FUNCTION_BLOCK integEC (* Basic Function Block Type *)
  (* Standard: 61499-2 *)
  (* Version 0.0, 2007-06-14, milos, nxtControl GmbH, Template *)
  PACKAGE Main;
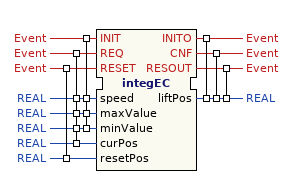
  EVENT_INPUT
    INIT WITH speed, maxValue, minValue; (* Initialization Request *)
    REQ WITH speed, maxValue, minValue, curPos; (* cycle calculation call *)
    RESET WITH resetPos;
  END_EVENT
  EVENT_OUTPUT
    INITO WITH liftPos; (* Initialization Confirm *)
    CNF WITH liftPos; (* Execution Confirmation *)
    RESOUT WITH liftPos;
  END_EVENT
  VAR_INPUT
    speed : REAL := 0.0; (* pv1 to integrate *)
    maxValue : REAL;
    minValue : REAL;
    curPos : REAL;
    resetPos : REAL;
  END_VAR
  VAR_OUTPUT
    liftPos : REAL := 0.0; (* out value (depends on integType) *)
  END_VAR
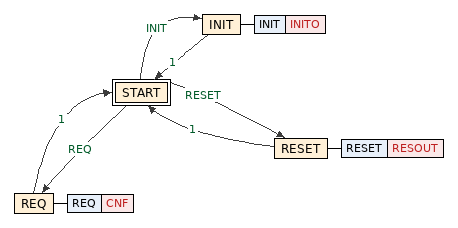
  EC_STATES
    START; (* Initial State *)
    INIT : INIT -> INITO; (* Initialization *)
    REQ : REQ -> CNF; (* Normal execution *)
    RESET : RESET -> RESOUT;
  END_STATES
  EC_TRANSITIONS
    START TO RESET := RESET;
    RESET TO START := 1;
    START TO REQ := REQ;
    REQ TO START := 1;
    START TO INIT := INIT;
    INIT TO START := 1;
  END_TRANSITIONS
  ALGORITHM INIT IN ST: (* Initialization algorithm *)
liftPos := 30.0;
  END_ALGORITHM
  ALGORITHM REQ IN ST:
liftPos := LIMIT(minValue, liftPos + speed, maxValue);
  END_ALGORITHM
  ALGORITHM RESET IN ST:
liftPos := resetPos;
  END_ALGORITHM
END_FUNCTION_BLOCK
